{attribute 'qualified_only'}
{attribute 'strict'}
{attribute 'to_string'}
TYPE E_CraneModes :
(
	Manual := 0,
	Auto := 1
);
END_TYPE

(* stored: Version 1.1.0.1, ProductVersion 3.1.4026.12
   DUT E_CraneModes: Id {941efdb5-96a6-4ada-830e-5d863ddd79f1} *)
